(* PLC project Magnet_Measurement, Beckhoff Automation GmbH TwinCAT PLC Control 3.5.13.21 *)
(* stored: creationDateTime 2023-11-09T09:08:17.7032943, modificationDateTime 2023-11-09T09:08:17.7032943 *)

PROGRAM Log_Data
VAR
	voltage_effective : REAL;
	voltage_frequency : REAL;
	current_effective : REAL;
	current_frequency : REAL;
	power : REAL;
    fbGetCurTaskIdx  : GETCURTASKINDEX;
    ncycletime       : UDINT;
	stDatabase : ST_Data;

	nState : INT;
	fb_PLCDBWriteEvt: FB_PLCDBWriteEvt(sNetID:='', tTimeout:=T#5S);
	arrColumns: ARRAY [0..2] OF STRING(50) := ['power', 'test', 'timestamp'];
	ipTcResult: Tc3_Database.I_TcMessage;
	sSourcePath: Tc3_Database.I_TcMessage;
	
END_VAR

            //// Convert Data and get the raw data
//voltage_effective := INT_TO_REAL(GVL_IO.gl_voltage_effective_raw)/65535*20; // Measured with an 
//voltage_frequency := 1/(UINT_TO_REAL(GVL_IO.gl_voltage_periode_raw)/1000); //convert ms to s and get Frequency from Period

//current_effective := INT_TO_REAL(GVL_IO.gl_current_effective_raw)/65535*20; // Measured with an 
//current_frequency := 1/(UINT_TO_REAL(GVL_IO.gl_current_periode_raw)/1000); //convert ms to s and get Frequency from Period

//fbGetCurTaskIdx();
//ncycletime := _TaskInfo[fbGetCurTaskIdx.index].CycleTime/10000;
//stDatabase.power := voltage_effective;
//stDatabase.test := current_effective;
//stDatabase.timestamp := timestamp;

//CASE nState OF
//	0: //Idle
//		;
//	1: //write
//		timestamp := index * ncycletime;
//		index := index + 1;
//		fb_PLCDBWriteEvt.WriteStruct(
//			hDBID:= 1, 
//			sTableName:= 'Magnet', 
//			pRecord:= ADR(stDatabase), 
//			cbRecord:= SIZEOF(stDatabase), 
//			pColumnNames:= ADR(arrColumns), 
//			cbColumnNames:= SIZEOF(arrColumns));
			
//		IF NOT fb_PLCDBWriteEvt.bBusy THEN
//			ipTcResult := fb_PLCDBWriteEvt.ipTcResult;
//			IF NOT fb_PLCDBWriteEvt.bError THEN
//				nState := 1;
//			ELSE
//				nState := 200;
//			END_IF
//		END_IF
//	200: //Event State
//		sSourcePath := ipTcResult;
//		nState := 0;
		
//		;
//END_CASE
          
END_PROGRAM
